TYPE EL2574_IO_Control_Color :
	STRUCT
		Red	  : USINT;
		Green : USINT;
		Blue  : USINT;
		White : USINT;
	END_STRUCT
END_TYPE

(* stored: Version 1.1.0.1, ProductVersion 3.1.4026.18
   DUT EL2574_IO_Control_Color: Id {2ab37f33-7c5d-4fff-b681-da78fc2247a0} *)
